SUBAPPLICATION mapping_Uebung_003b2 (* Funk 16 Tasten auf DataPanel 16 *)
  (* Standard: 61499-2; Description: Copyright (c) 2023 Meisterschulen am Ostbahnhof This program and the accompanying materials are made available under the terms of the Eclipse Public License 2.0 which is available at https://www.eclipse.org/legal/epl-2.0/ SPDX-License-Identifier: EPL-2.0 *)
  (* Version 1.0, 2023-10-23, Franz Höpfinger, Meisterschulen am Ostbahnhof *)
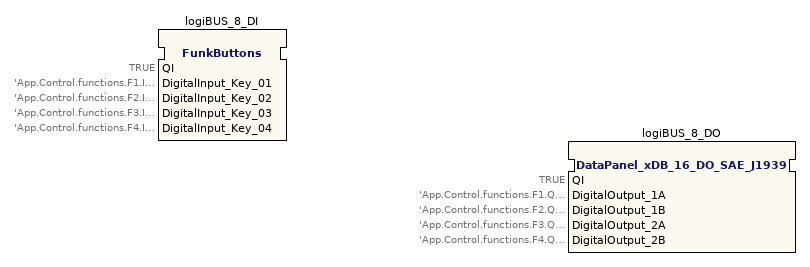
  FBS
    logiBUS_8_DO : DataPanel_xDB_16_DO_SAE_J1939(QI := TRUE, DigitalOutput_1A := 'App.Control.functions.F1.QX', DigitalOutput_1B := 'App.Control.functions.F2.QX', DigitalOutput_2A := 'App.Control.functions.F3.QX', DigitalOutput_2B := 'App.Control.functions.F4.QX');
    logiBUS_8_DI : FunkButtons(QI := TRUE, DigitalInput_Key_01 := 'App.Control.functions.F1.IX', DigitalInput_Key_02 := 'App.Control.functions.F2.IX', DigitalInput_Key_03 := 'App.Control.functions.F3.IX', DigitalInput_Key_04 := 'App.Control.functions.F4.IX');
  END_FBS
END_SUBAPPLICATION
